{attribute 'GeneratedUsingTerminal: EP2816-0008-0016'}
{attribute addProperty BoxType "EP2816-0008-0016"}
{attribute addProperty Id "Diag_InputAT %I*ARRAY[0..7] OF BOOL8"}
{attribute addProperty CRC "568896300"}
{attribute addProperty Size "8"}
TYPE DO_Inputs_Channel_584303BF :
STRUCT
	{attribute addProperty Name "Diag_Input"}
	Diag_Input AT %I* : ARRAY[0..7] OF BOOL;
END_STRUCT
END_TYPE

(* stored: Version 1.2.0.0, ProductVersion 3.1.4024.9
   DUT DO_Inputs_Channel_584303BF: Id {2977aa29-d8e4-42cf-8a9f-bc6bd264729c} *)
